{attribute 'qualified_only'}
VAR_GLOBAL
	uniDO : uni_OutputModule;
END_VAR

(* stored: Version 1.1.0.1, ProductVersion 3.1.4024.13
   GVL GVL_Output: Id {53a41dba-fec7-41ec-9c76-66996f1278ba} *)
